FUNCTION_BLOCK FutureMCHaltCreator IMPLEMENTS InterfaceTaskCreator
VAR_INPUT
END_VAR
VAR_OUTPUT
END_VAR
VAR
	_axis: REFERENCE TO AXIS_REF;
	_deceleration: MC_LREAL;
	_jerk		: MC_LREAL;
	_option : ST_MoveOptions;
	_buffer_mode : MC_BufferMode;
END_VAR

{warning 'add method implementation '}
METHOD create_future : InterfaceFuture
VAR_INPUT
	(* Specify future name*)
	future_name	: STRING;
END_VAR
VAR
	_p_future : POINTER TO FutureMCHalt;
END_VAR
_p_future := __NEW(FutureMCHalt);
_p_future^.future_name := future_name;
_p_future^.set_parameters(_axis, _deceleration, _jerk);
_p_future^.set_options(_buffer_mode, _option);
create_future := _p_future^;
END_METHOD

{warning 'add method implementation '}
METHOD destroy_future : InterfaceFuture
VAR_INPUT
	(* Specify future instance whtat you want to delete.*)
	future	: InterfaceFuture;
END_VAR
VAR
	_p_future : POINTER TO FutureMCHalt;
END_VAR
IF __QUERYPOINTER(future, _p_future) THEN
	__DELETE(_p_future);
	IF _p_future = 0  THEN
		destroy_future := 0;
	END_IF
END_IF
END_METHOD

METHOD set_options : BOOL
VAR_INPUT
	buffer_mode : MC_BufferMode;
	option : ST_MoveOptions;
END_VAR
_buffer_mode := buffer_mode;
_option := option;
END_METHOD

METHOD set_parameters : BOOL
VAR_INPUT
	axis : REFERENCE TO AXIS_REF;
	deceleration	: MC_LREAL;		// Set deceleration in case let moving axis halt.
	jerk			: MC_LREAL;		// Set jerk in case let moving axis halt.
END_VAR
_axis REF= axis;
_deceleration := deceleration;
_jerk := jerk;
END_METHOD

END_FUNCTION_BLOCK

(* stored: Version 1.1.0.1, ProductVersion 3.1.4024.15
   POU FutureMCHaltCreator: Id {c70f48d7-b1d0-4e9a-ac25-e3539499ee8d}, SpecialFunc None
   Method create_future: Id {b5dcb4f1-25ee-4051-a78b-2c288ff5a3c3}
   Method destroy_future: Id {58754b79-06fa-4918-8569-eecf49c52cff}
   Method set_options: Id {525cc8ff-850d-4432-a941-cc9fce4f6d10}
   Method set_parameters: Id {3dd5dd28-dfd6-499a-adc2-52c4b43f7a24} *)
